(* CODESYS project CFC_FB.pou_xml.xml

Project tree, tasks and I/O mapping:
  function block CFC_FB [CFC]
*)

// CFC_FB
FUNCTION_BLOCK CFC_FB
VAR_INPUT
END_VAR
VAR_OUTPUT
END_VAR
VAR
	auxBool : BOOL;
	CLK : BOOL;
	R_TRIG_OUT : BOOL;
END_VAR
VAR // added by the converter: edge detectors and wires of the graphical bodies
    _w1 : ANY;
END_VAR

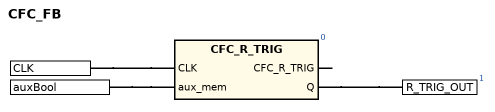
CFC_R_TRIG(CLK := CLK, aux_mem := auxBool, Q => _w1);
R_TRIG_OUT := _w1;

END_FUNCTION_BLOCK
